(* CODESYS project GomelChemical_2PLC.export

Project tree, tasks and I/O mapping:
  application Application
    libraries: 
    task PLC_Task (cyclic, interval t#50ms, priority 15) calls PLC_PRG
    GV/
      global variables _DO
      global variables AI
      global variables DI
      global variables HMI_Ons
      global variables HMI_Sensors
      global variables HMI_Settings
    IO/
      Device/
        program prOnOff [ST]
      program prAItoValue [ST]
      program prInToVars [ST]
      program prVarsToOut [ST]
    program PLC_PRG [ST]
*)

// Application/GV/_DO

VAR_GLOBAL
	DO_IgniteFurbece_120			: BOOL;
	DO_GasValveHSV46_120			: BOOL;
	DO_GasValveHSV47_120			: BOOL;
	DO_GasValveHSV48				: BOOL;
	DO_GasValveHSV49_120			: BOOL;
	DO_H2SO4ValveHSV205S_102		: BOOL;
	DO_Vent_35A_35B					: BOOL;
	DO_NH3valve_HZSV140				: BOOL;
	DO_LightAlmGranul_HL300_1		: BOOL;
	DO_SoundAlmGranul_HA300_1		: BOOL;
	DO_LightAlmGranul_HL300_2		: BOOL;
	DO_SoundAlmGranul_HA300_2		: BOOL;
	DO_LightAlmReact_100_HL300_3	: BOOL;
	DO_SoundAlmReact_100_HA300_3	: BOOL;
	DO_SoundAlm_HA1					: BOOL;
	DO_SoundAlm_HA2					: BOOL;
	DO_ExhaustVent_35_A_B			: BOOL;
	
	
	//////////////////////////////////////////////////////////
	
	
	_DO_IgniteFurbece_120		: BOOL;
_DO_GasValveHSV46_120			: BOOL;
_DO_GasValveHSV47_120			: BOOL;
_DO_GasValveHSV48				: BOOL;
_DO_GasValveHSV49_120			: BOOL;
_DO_H2SO4ValveHSV205S_102		: BOOL;
_DO_Vent_35A_35B				: BOOL;
_DO_NH3valve_HZSV140			: BOOL;
_DO_LightAlmGranul_HL300_1		: BOOL;
_DO_SoundAlmGranul_HA300_1		: BOOL;
_DO_LightAlmGranul_HL300_2		: BOOL;
_DO_SoundAlmGranul_HA300_2		: BOOL;
_DO_LightAlmReact_100_HL300_3	: BOOL;
_DO_SoundAlmReact_100_HA300_3	: BOOL;
_DO_SoundAlm_HA1				: BOOL;
_DO_SoundAlm_HA2				: BOOL;
_DO_ExhaustVent_35_A_B			: BOOL;


	
	
END_VAR

// Application/GV/AI

VAR_GLOBAL
	AI_HN3PressInZech_PZIRA1_1					: INT;	
	AI_HN3PressBeforeTubeReact_100_PZIRA2_1		: INT;
	AI_HN3PressBeforeTubeReact_100_1_PZIRA2_2	: INT;
	AI_HN3ConcInAirInGranul_QZIRA3_1			: INT;
	
	
	///////////////////////////////////////////////////////////////
	
	
	_AI_HN3PressInZech_PZIRA1_1					: INT;
	_AI_HN3PressBeforeTubeReact_100_PZIRA2_1	: INT;
	_AI_HN3PressBeforeTubeReact_100_1_PZIRA2_2	: INT;
	_AI_HN3ConcInAirInGranul_QZIRA3_1			: INT;

END_VAR

// Application/GV/DI

VAR_GLOBAL
	DI_HSV47_Opn	: BOOL;
	DI_HSV47_Cls	: BOOL;
	DI_HSV205_Opn	: BOOL;
	DI_HSV205_Cls	: BOOL;
	DI_HSVZ140_Opn	: BOOL;
	DI_HSVZ140_Cls	: BOOL;
	DI_VentWorking_35A	: BOOL;
	DI_VentWorking_35B	: BOOL;
	
	
	
	/////////////////////////////////////
	
	
	_DI_HSV47_Opn	: BOOL;
	_DI_HSV47_Cls	: BOOL;
	_DI_HSV205_Opn	: BOOL;
	_DI_HSV205_Cls	: BOOL;
	_DI_HSVZ140_Opn	: BOOL;
	_DI_HSVZ140_Cls	: BOOL;
	_DI_VentWorking_35A	: BOOL;
	_DI_VentWorking_35B	: BOOL;

	
END_VAR

// Application/GV/HMI_Ons

VAR_GLOBAL
	IgniteFurbece_120			: BOOL;
	GasValveHSV46_120			: BOOL;
	GasValveHSV47_120			: BOOL;
	GasValveHSV48				: BOOL;
	GasValveHSV49_120			: BOOL;
	H2SO4ValveHSV205S_102		: BOOL;
	Vent_35A_35B				: BOOL;
	NH3valve_HZSV140			: BOOL;
	LightAlmGranul_HL300_1		: BOOL;
	SoundAlmGranul_HA300_1		: BOOL;
	LightAlmGranul_HL300_2		: BOOL;
	SoundAlmGranul_HA300_2		: BOOL;
	LightAlmReact_100_HL300_3	: BOOL;
	SoundAlmReact_100_HA300_3	: BOOL;
	SoundAlm_HA1				: BOOL;
	SoundAlm_HA2				: BOOL;
	ExhaustVent_35_A_B			: BOOL;

END_VAR

// Application/GV/HMI_Sensors

VAR_GLOBAL
	HN3PressInZech_PZIRA1_1						: REAL;
	HN3PressBeforeTubeReact_100_PZIRA2_1		: REAL;
	HN3PressBeforeTubeReact_100_1_PZIRA2_2		: REAL;
	HN3ConcInAirInGranul_QZIRA3_1				: REAL;

END_VAR

// Application/GV/HMI_Settings

VAR_GLOBAL
	HN3PressInZech_PZIRA1_1_CalCoef	: REAL:=1;
HN3PressBeforeTubeReact_100_PZIRA2_1_CalCoef	: REAL:=1;
HN3PressBeforeTubeReact_100_1_PZIRA2_2_CalCoef	: REAL:=1;
HN3ConcInAirInGranul_QZIRA3_1_CalCoef	: REAL:=1;


HN3PressInZech_PZIRA1_1_Offset	: REAL;
HN3PressBeforeTubeReact_100_PZIRA2_1_Offset	: REAL;
HN3PressBeforeTubeReact_100_1_PZIRA2_2_Offset	: REAL;
HN3ConcInAirInGranul_QZIRA3_1_Offset	: REAL;


END_VAR

// Application/PLC_PRG
PROGRAM PLC_PRG
VAR
END_VAR

prInToVars();
prAItoValue();
prAItoValue();
prVarsToOut();

END_PROGRAM

// Application/IO/prInToVars
PROGRAM prInToVars
VAR
END_VAR

DI_HSV47_Opn	:=	_DI_HSV47_Opn	;
DI_HSV47_Cls	:=	_DI_HSV47_Cls	;
DI_HSV205_Opn	:=	_DI_HSV205_Opn	;
DI_HSV205_Cls	:=	_DI_HSV205_Cls	;
DI_HSVZ140_Opn	:=	_DI_HSVZ140_Opn	;
DI_HSVZ140_Cls	:=	_DI_HSVZ140_Cls	;
DI_VentWorking_35A	:=	_DI_VentWorking_35A	;
DI_VentWorking_35B	:=	_DI_VentWorking_35B	;


AI_HN3PressInZech_PZIRA1_1	:=	_AI_HN3PressInZech_PZIRA1_1	;
AI_HN3PressBeforeTubeReact_100_PZIRA2_1	:=	_AI_HN3PressBeforeTubeReact_100_PZIRA2_1	;
AI_HN3PressBeforeTubeReact_100_1_PZIRA2_2	:=	_AI_HN3PressBeforeTubeReact_100_1_PZIRA2_2	;
AI_HN3ConcInAirInGranul_QZIRA3_1	:=	_AI_HN3ConcInAirInGranul_QZIRA3_1	;

END_PROGRAM

// Application/IO/prAItoValue
PROGRAM prAItoValue
VAR
END_VAR

HN3PressInZech_PZIRA1_1:=AI_TO_Current(AI_HN3PressInZech_PZIRA1_1) *HN3PressInZech_PZIRA1_1_CalCoef  +HN3PressInZech_PZIRA1_1_Offset;
HN3PressBeforeTubeReact_100_PZIRA2_1:=AI_TO_Current(AI_HN3PressBeforeTubeReact_100_PZIRA2_1) *HN3PressBeforeTubeReact_100_PZIRA2_1_CalCoef  +HN3PressBeforeTubeReact_100_PZIRA2_1_Offset;
HN3PressBeforeTubeReact_100_1_PZIRA2_2:=AI_TO_Current(AI_HN3PressBeforeTubeReact_100_1_PZIRA2_2) *HN3PressBeforeTubeReact_100_1_PZIRA2_2_CalCoef  +HN3PressBeforeTubeReact_100_1_PZIRA2_2_Offset;
HN3ConcInAirInGranul_QZIRA3_1:=AI_TO_Current(AI_HN3ConcInAirInGranul_QZIRA3_1) *HN3ConcInAirInGranul_QZIRA3_1_CalCoef  +HN3ConcInAirInGranul_QZIRA3_1_Offset;

END_PROGRAM

// Application/IO/prVarsToOut
PROGRAM prVarsToOut
VAR
END_VAR

_DO_IgniteFurbece_120	:=	DO_IgniteFurbece_120	;
_DO_GasValveHSV46_120	:=	DO_GasValveHSV46_120	;
_DO_GasValveHSV47_120	:=	DO_GasValveHSV47_120	;
_DO_GasValveHSV48	:=	DO_GasValveHSV48	;
_DO_GasValveHSV49_120	:=	DO_GasValveHSV49_120	;
_DO_H2SO4ValveHSV205S_102	:=	DO_H2SO4ValveHSV205S_102	;
_DO_Vent_35A_35B	:=	DO_Vent_35A_35B	;
_DO_NH3valve_HZSV140	:=	DO_NH3valve_HZSV140	;
_DO_LightAlmGranul_HL300_1	:=	DO_LightAlmGranul_HL300_1	;
_DO_SoundAlmGranul_HA300_1	:=	DO_SoundAlmGranul_HA300_1	;
_DO_LightAlmGranul_HL300_2	:=	DO_LightAlmGranul_HL300_2	;
_DO_SoundAlmGranul_HA300_2	:=	DO_SoundAlmGranul_HA300_2	;
_DO_LightAlmReact_100_HL300_3	:=	DO_LightAlmReact_100_HL300_3	;
_DO_SoundAlmReact_100_HA300_3	:=	DO_SoundAlmReact_100_HA300_3	;
_DO_SoundAlm_HA1	:=	DO_SoundAlm_HA1	;
_DO_SoundAlm_HA2	:=	DO_SoundAlm_HA2	;
_DO_ExhaustVent_35_A_B	:=	DO_ExhaustVent_35_A_B	;

END_PROGRAM

// Application/IO/Device/prOnOff
PROGRAM prOnOff
VAR
END_VAR

DO_IgniteFurbece_120	:=	IgniteFurbece_120	;
DO_GasValveHSV46_120	:=	GasValveHSV46_120	;
DO_GasValveHSV47_120	:=	GasValveHSV47_120	;
DO_GasValveHSV48		:=	GasValveHSV48	;
DO_GasValveHSV49_120	:=	GasValveHSV49_120	;
DO_H2SO4ValveHSV205S_102	:=	H2SO4ValveHSV205S_102	;
DO_Vent_35A_35B	:=	Vent_35A_35B	;
DO_NH3valve_HZSV140	:=	NH3valve_HZSV140	;
DO_LightAlmGranul_HL300_1	:=	LightAlmGranul_HL300_1	;
DO_SoundAlmGranul_HA300_1	:=	SoundAlmGranul_HA300_1	;
DO_LightAlmGranul_HL300_2	:=	LightAlmGranul_HL300_2	;
DO_SoundAlmGranul_HA300_2	:=	SoundAlmGranul_HA300_2	;
DO_LightAlmReact_100_HL300_3	:=	LightAlmReact_100_HL300_3	;
DO_SoundAlmReact_100_HA300_3	:=	SoundAlmReact_100_HA300_3	;
DO_SoundAlm_HA1	:=	SoundAlm_HA1	;
DO_SoundAlm_HA2	:=	SoundAlm_HA2	;
DO_ExhaustVent_35_A_B	:=	ExhaustVent_35_A_B	;

END_PROGRAM
